	                ///////////// 1660: chiusura chela lato 2 (HMI)
	            1660:
	                "DB_RobotMission".Gripper_Side := 2;
	                "DB_RobotMission".Gripper_code := #Gripper_ID[2];
	                "DB_RobotMission".Command := "CMD_RobotCloseGripper2";
	                #Dispatcher["_master"] := 1661;
	            1661:
	                IF "DB_RobotMissionStatus".StatusCode = "cmd_acquired" OR
	                    "DB_RobotMissionStatus".StatusCode = "cmd_executing" THEN
	                    #Dispatcher["_master"] := 1662;
	                END_IF;
	            1662:
	                IF "DB_RobotMissionStatus".StatusCode = "cmd_executed" THEN
	                    "DB_RobotMission".Command := 0;
	                    #MissionCode := 0;
	                    #Dispatcher["_master"] := 0;
	                END_IF;
	                ///////////// 1700: posizionamento davanti a MC1 (automatico)
	                // Il robot si porta in attesa e la missione chiude: restera' fermo
	                // li' perche' FB204 non assegna nulla finche' la porta non si apre.
	            1700:
	                IF "DB_RobotMissionStatus".StatusCode = "cmd_acquired" OR
	                    "DB_RobotMissionStatus".StatusCode = "cmd_executing" THEN
	                    #Dispatcher["_master"] := 1701;
	                ELSIF "DB_RobotMissionStatus".StatusCode = "cmd_rejected" OR
	                    "DB_RobotMissionStatus".StatusCode = "cmd_aborted" THEN
	                    "DB_RobotMission".Command := 0;
	                    #Error := "MISSION_PositioningMC_AUTO" * 100 + 22;
	                    #MissionCode := 0;
	                    #Dispatcher["_master"] := 0;
	                END_IF;
	            1701:
	                IF "DB_RobotMissionStatus".StatusCode = "cmd_executed" THEN
	                    "DB_RobotMission".Command := 0;
	                    #MissionCode := 0;
	                    #Dispatcher["_master"] := 0;
	                END_IF;
	                ///////////// 1750: ritorno in home (automatico)
	                // Stessa struttura del 1700: attesa acquisizione con gestione del
	                // rifiuto, poi attesa esecuzione. Il robot ci va e resta li'.
	            1750:
	                IF "DB_RobotMissionStatus".StatusCode = "cmd_acquired" OR
	                    "DB_RobotMissionStatus".StatusCode = "cmd_executing" THEN
	                    #Dispatcher["_master"] := 1751;
	                ELSIF "DB_RobotMissionStatus".StatusCode = "cmd_rejected" OR
	                    "DB_RobotMissionStatus".StatusCode = "cmd_aborted" THEN
	                    // il robot non ha accettato: si chiude comunque. Il home e' una
	                    // rifinitura, non deve fermare la cella se fallisce.
	                    "DB_RobotMission".Command := 0;
	                    #MissionCode := 0;
	                    #Dispatcher["_master"] := 0;
	                END_IF;
	            1751:
	                IF "DB_RobotMissionStatus".StatusCode = "cmd_executed" THEN
	                    "DB_RobotMission".Command := 0;
	                    #MissionCode := 0;
	                    #Dispatcher["_master"] := 0;
	                END_IF;
	        END_CASE;
	    END_IF;

	END_REGION

	REGION Gripper_MANAGER
	    REGION Gripper_Robot_to_TRAY
	        CASE #Dispatcher["_Gripper_Robot_to_TRAY"] OF
	            0:  //nothing to do
	                ;
	            10:  //prepare mission data
	                IF "SqlCommands".sqlCommands[0] = '' THEN
	                    IF NOT "DB_BOX_1".Robot_enabled_to_work THEN
	                        #Error := 949;
	                        #Dispatcher["_Gripper_Robot_to_TRAY"] := 0;
	                    ELSE
	                        #queryTemp := CONCAT(IN1 := 'SELECT X,Y,Z,X_ROT,Y_ROT,Z_ROT,APPROACH_TYPE,APPROACH_X,APPROACH_Y,APPROACH_Z from COORDINATES_GRIPPER_SHELF where id=',
	                                             IN2 := "INT_TO_STRING_WITHOUT_SIGN"(#Gripper_ID[1]));
	                        #queryStartExecution := TRUE;

	                        #Dispatcher["_Gripper_Robot_to_TRAY"] := 20;
	                    END_IF;
	                END_IF;

	            20:  // wait for result DB -> prepare mission data
	                // PRESA IN CARICO VERIFICATA: SqlData e' un buffer unico condiviso,
	                // senza il confronto su sqlCommands[0] si legge la risposta di un
	                // altro richiedente — qui sarebbe lo SLOT A SCAFFALE dove posare
	                // la pinza.
	                IF NOT "DB_executeQuery".readyForNextQuery
	                    AND "SqlCommands".sqlCommands[0] = #queryTemp THEN
	                    #Dispatcher["_Gripper_Robot_to_TRAY"] := 25;
	                END_IF;

	            25: //execute query
	                IF "DB_executeQuery".dataReady AND "DB_executeQuery".noData THEN
	                    // slot di casa della pinza non trovato a scaffale: con FB6
	                    // corretto "zero righe" non e' piu' dataError, va preso qui.
	                    #Error := 990;
	                    "DB_executeQuery".readyForNextQuery := TRUE;
	                    #Dispatcher["_Gripper_Robot_to_TRAY"] := 990;
	                ELSIF "DB_executeQuery".dataReady AND NOT "DB_executeQuery".dataError THEN

	                    "DB_RobotMission".Command := "CMD_RobotRemoveGripper";
	                    "DB_RobotMission"."X_Pick-Place" := "SqlData".data.rows[0].col[0];
	                    "DB_RobotMission"."Y_Pick-Place" := "SqlData".data.rows[0].col[1];
	                    "DB_RobotMission"."Z_Pick-Place" := "SqlData".data.rows[0].col[2];
	                    "DB_RobotMission"."XRot_Pick-Place" := "SqlData".data.rows[0].col[3];
	                    "DB_RobotMission"."YRot_Pick-Place" := "SqlData".data.rows[0].col[4];
	                    "DB_RobotMission"."ZRot_Pick-Place" := "SqlData".data.rows[0].col[5];
	                    "DB_RobotMission".X_approach := "SqlData".data.rows[0].col[7];
	                    "DB_RobotMission".Y_approach := "SqlData".data.rows[0].col[8];
	                    "DB_RobotMission".Z_approach := "SqlData".data.rows[0].col[9];
	                    "DB_RobotMission".XRot_approach := 0;
	                    "DB_RobotMission".YRot_approach := 0;
	                    "DB_RobotMission".ZRot_approach := 0;
	                    //"DB_RobotMission".ApproachType := DINT_TO_INT("SqlData".data.rows[0].col[6]);
	                    "DB_RobotMission".ApproachType := "FC_ExtractApproach"(approachVal := "SqlData".data.rows[0].col[6], pick := FALSE);
	                    "DB_RobotMission".Object_Type := "Gripper";
	                    "DB_RobotMission".Unit_code := "Warehouse1";
	                    "DB_RobotMission".Gripper_code := #Gripper_ID[1];
	                    //"DB_RobotMission".Option

	                    "DB_executeQuery".readyForNextQuery := TRUE;

	                    #Dispatcher["_Gripper_Robot_to_TRAY"] := 30;
	                ELSIF "DB_executeQuery".dataError THEN
	                    // Alarm
	                    #Error := 990;
	                    "DB_executeQuery".readyForNextQuery := TRUE;

	                    #Dispatcher["_Gripper_Robot_to_TRAY"] := 990;
	                END_IF;
	            30:  // start robot mission
	                //"DB_RobotMission".Command := "CMD_RobotRemoveGripper";
	                IF "DB_RobotMissionStatus".StatusCode = "cmd_acquired" OR
	                    "DB_RobotMissionStatus".StatusCode = "cmd_executing" THEN
	                    #Dispatcher["_Gripper_Robot_to_TRAY"] := 40;
	                END_IF;
	            40:  // finished -> update DB
	                // DOPPIA CONFERMA (5/9), simmetrica a quella del carico allo
	                // stato 50 di Gripper_TRAY_to_Robot: non basta cmd_executed del
	                // robot, serve anche che il sensore NON veda piu' la pinza.
	                // Senza, i registri direbbero "flangia nuda" con la pinza ancora
	                // attaccata, e ogni scelta successiva partirebbe da un dato falso.
	                // Stallo qui = guardare %I502.0.
	                // NB: lo scarico NON passa dalla catena unica — azzerare i registri
	                // e' un gesto che non ha bisogno di cercare gemelle, e #GripperRequested
	                // deve restare intatto per il carico che i rami 110/210/310/410/510
	                // lanciano subito dopo.
	                IF "DB_RobotMissionStatus".StatusCode = "cmd_executed"
	                    AND NOT "Gripper_mounted"
	                THEN
	                    "DB_RobotMission".Command := 0;  ///\\\
	                    #Gripper_ID[1] := 0;
	                    #Gripper_ID[2] := 0;
	                    #Dispatcher["updateGripperOnRobot"] := 10;

	                    #Dispatcher["_Gripper_Robot_to_TRAY"] := 50;
	                END_IF;
	            50: // attesa fine update DB -> chiusura catena scarico
	                IF #Dispatcher["updateGripperOnRobot"] = 0 THEN
	                    #Dispatcher["_Gripper_Robot_to_TRAY"] := 0;
	                END_IF;

	        END_CASE;
	    END_REGION

	    REGION Gripper_TRAY_to_Robot
	        CASE #Dispatcher["_Gripper_TRAY_to_Robot"] OF
	            0: // nothing to do
	                ;
	            10: //prepare mission data
	                IF "SqlCommands".sqlCommands[0] = '' THEN
	                    IF NOT "DB_BOX_1".Robot_enabled_to_work THEN
	                        #Error := 949;
	                        #Dispatcher["_Gripper_TRAY_to_Robot"] := 0;
	                    ELSE
	                        // SORGENTE UNICA: #GripperRequested (17/9).
	                        // Prima i tre rami leggevano sorgenti diverse — GripperRequested
	                        // per il magazzino, order.GRIPPER per MC1, order.GRIPPER di MC1
	                        // anche nel ramo MC2 (refuso). Nel ciclo automatico i valori
	                        // coincidono perche' i master 100/300/400/500 scrivono
	                        // GripperRequested := order.GRIPPER prima di lanciare, ma
	                        // l'accoppiamento era implicito: la catena cercava a scaffale
	                        // una pinza e la catena unica ne registrava un'altra se le due
	                        // sorgenti divergevano.
	                        // Adesso chi lancia dice QUALE pinza vuole, e questa catena
	                        // la cerca e basta — stessa variabile che _Set_Gripper_OnBoard
	                        // usera' per scrivere i registri.
	                        IF #GripperRequested > 0 THEN
	                            // GEMELLA SOLO CON SUB_POS VALORIZZATO (5/10, concordato 1/9): una pinza
	                            // singola ha SUB_POS = 0, e "SUB_POS in (0)" tirava dentro tutte le altre
	                            // pinze singole a scaffale come se fossero il suo lato 2.
	                            #queryTemp := CONCAT_STRING(IN1 := 'select X,Y,Z,X_rot,Y_rot,Z_ROT, APPROACH_TYPE, APPROACH_X, APPROACH_Y, APPROACH_Z, ID from COORDINATES_GRIPPER_SHELF where id=',
	                                                        IN2 := "INT_TO_STRING_WITHOUT_SIGN"(#GripperRequested),
	                                                        IN3 := ' OR (SUB_POS>0 AND SUB_POS in (select sub_pos from COORDINATES_GRIPPER_SHELF where id=',
	                                                        IN4 := "INT_TO_STRING_WITHOUT_SIGN"(#GripperRequested),
	                                                        IN5 := ')) order by gripper_sub_pos');
	                            #queryStartExecution := TRUE;
	                            #Dispatcher["_Gripper_TRAY_to_Robot"] := 20;
	                        ELSE
	                            // nessuna pinza richiesta: senza questa guardia la query
	                            // usciva con id=0, zero righe e 990 — lo stesso difetto
	                            // che il 17/9 ha tenuto appeso il master ai rami 1xx.
	                            #Error := 937;   // pinza target non valida
	                            #Dispatcher["_Gripper_TRAY_to_Robot"] := 0;
	                        END_IF;
	                    END_IF;
	                END_IF;

	            20:  //execute query
	                // PRESA IN CARICO VERIFICATA: SqlData e' un buffer unico condiviso,
	                // senza il confronto su sqlCommands[0] si legge la risposta di un
	                // altro richiedente — qui sarebbe lo SLOT della pinza da prendere.
	                IF NOT "DB_executeQuery".readyForNextQuery
	                    AND "SqlCommands".sqlCommands[0] = #queryTemp THEN
	                    #Dispatcher["_Gripper_TRAY_to_Robot"] := 30;
	                END_IF;

	            30: // wait anwser
	                IF "DB_executeQuery".dataReady AND "DB_executeQuery".noData THEN
	                    // pinza richiesta non trovata a scaffale. Ramo NUOVO: prima
	                    // non esisteva, e con FB6 corretto la catena proseguirebbe
	                    // con coordinate a zero mandando il robot a sbattere.
	                    #Error := 990;
	                    "DB_executeQuery".readyForNextQuery := true;
	                    #Dispatcher["_Gripper_TRAY_to_Robot"] := 0;
	                ELSIF "DB_executeQuery".dataReady AND NOT "DB_executeQuery".dataError THEN
	                    "DB_RobotMission"."X_Pick-Place" := "SqlData".data.rows[0].col[0];
	                    "DB_RobotMission"."Y_Pick-Place" := "SqlData".data.rows[0].col[1];
	                    "DB_RobotMission"."Z_Pick-Place" := "SqlData".data.rows[0].col[2];
	                    "DB_RobotMission"."XRot_Pick-Place" := "SqlData".data.rows[0].col[3];
	                    "DB_RobotMission"."YRot_Pick-Place" := "SqlData".data.rows[0].col[4];
	                    "DB_RobotMission"."ZRot_Pick-Place" := "SqlData".data.rows[0].col[5];
	                    "DB_RobotMission".X_approach := "SqlData".data.rows[0].col[7];
	                    "DB_RobotMission".Y_approach := "SqlData".data.rows[0].col[8];
	                    "DB_RobotMission".Z_approach := "SqlData".data.rows[0].col[9];
	                    "DB_RobotMission".XRot_approach := 0;
	                    "DB_RobotMission".YRot_approach := 0;
	                    "DB_RobotMission".ZRot_approach := 0;
	                    //"DB_RobotMission".ApproachType := DINT_TO_INT("SqlData".data.rows[0].col[6]);
	                    "DB_RobotMission".ApproachType := "FC_ExtractApproach"(approachVal := "SqlData".data.rows[0].col[6], pick := TRUE);
	                    "DB_RobotMission".Object_Type := "Gripper";
	                    "DB_RobotMission".Unit_code := "Warehouse1";
	                    "DB_RobotMission".Gripper_code := DINT_TO_INT(#GripperRequested);
	                    //"DB_RobotMission".Option

	                    // LATO 2 NON PIU' QUI (17/9): lo scrive la catena
	                    // _Set_Gripper_OnBoard, che e' il punto unico. Questo stato
	                    // leggeva le coordinate di prelievo e per comodita' anche la
	                    // gemella, ma quella doppia responsabilita' e' proprio il
	                    // motivo per cui lo swap — che non passa di qui — dimenticava
	                    // il lato 2.

	                    "DB_executeQuery".readyForNextQuery := true;

	                    #Dispatcher["_Gripper_TRAY_to_Robot"] := 40;
	                ELSIF "DB_executeQuery".dataError THEN
	                    // ramo NUOVO: errore vero del ponte
	                    #Error := 990;
	                    "DB_executeQuery".readyForNextQuery := true;
	                    #Dispatcher["_Gripper_TRAY_to_Robot"] := 0;
	                END_IF;

	            40:  // start Robot mission
	                IF "DB_RobotMissionStatus".StatusCode = "cmd_executed" OR
	                    "DB_RobotMissionStatus".StatusCode = "cmd_waitingNewCmd" THEN
	                    "DB_RobotMission".Command := "CMD_RobotPickGripper";

	                    #Dispatcher["_Gripper_TRAY_to_Robot"] := 45;
	                END_IF;
	            45:
	                //"DB_RobotMission".Command := "CMD_RobotPickGripper";
	                IF "DB_RobotMissionStatus".StatusCode = "cmd_acquired" OR
	                    "DB_RobotMissionStatus".StatusCode = "cmd_executing" THEN

	                    #Dispatcher["_Gripper_TRAY_to_Robot"] := 50;
	                END_IF;

	            50: // latch a doppia conferma: esito missione + sensore fisico — stallo qui = guardare %I502.0
	                IF "DB_RobotMissionStatus".StatusCode = "cmd_executed" AND "Gripper_mounted" THEN

	                    // AZZERAMENTO COMANDO (5/9): senza, il robot resta a
	                    // cmd_executed in attesa che il PLC risponda, e get_TCP_Data
	                    // allo stato 40 aspetta che il robot torni a waitingNewCmd:
	                    // stallo circolare col master fermo al 960.
	                    "DB_RobotMission".Command := 0;  ///\\\

	                    // registri + database alla catena unica (17/9)
	                    #Dispatcher["_Set_Gripper_OnBoard"] := 10;
	                    #Dispatcher["_Gripper_TRAY_to_Robot"] := 60;
	                END_IF;
	            60: // attesa fine registrazione -> chiusura catena carico
	                IF #Dispatcher["_Set_Gripper_OnBoard"] = 0 THEN
	                    #Dispatcher["_Gripper_TRAY_to_Robot"] := 0;
	                END_IF;
	        END_CASE;

	    END_REGION

	    REGION Gripper_Hook_Search
	        CASE #Dispatcher["_Gripper_Hook_Search"] OF
	            0: // nothing to do
	                ;
	            10: //prepare mission data
	                IF "SqlCommands".sqlCommands[0] = '' THEN
	                    //#queryTemp := 'select id,pos_mag-1000 from gripper where pos_mag>1000 and pos_plant>=0';
	                    #queryTemp := 'select id,sub_pos-1000 from gripper where sub_pos>1000 AND pos_plant>=0';
	                    #queryStartExecution := TRUE;
	                    #Dispatcher["_Gripper_Hook_Search"] := 20;
	                END_IF;

	            20:  //execute query
	                // PRESA IN CARICO VERIFICATA: SqlData e' un buffer unico condiviso,
	                // senza il confronto su sqlCommands[0] si legge la risposta di un
	                // altro richiedente — qui finirebbe in GripperRequested un ID pinza
	                // preso da una colonna qualsiasi di un'altra query.
	                IF NOT "DB_executeQuery".readyForNextQuery
	                    AND "SqlCommands".sqlCommands[0] = #queryTemp THEN
	                    #Dispatcher["_Gripper_Hook_Search"] := 30;
	                END_IF;

	            30: // wait anwser
	                IF "DB_executeQuery".dataReady THEN
	                    IF "DB_executeQuery".noData OR "DB_executeQuery".dataError THEN
	                        #Error := 22;
	                    ELSE
	                        #GripperRequested := DINT_TO_INT("SqlData".data.rows[0].col[1]);
	                    END_IF;

	                    "DB_executeQuery".readyForNextQuery := true;
	                    #Dispatcher["_Gripper_Hook_Search"] := 0;
	                END_IF;
	        END_CASE;

	    END_REGION

	    REGION Gripper4Pallet_Search
	        CASE #Dispatcher["_Gripper4Pallet_Search"] OF
	            0: // nothing to do
	                ;
	            10: //prepare mission data
	                IF "SqlCommands".sqlCommands[0] = '' THEN
	                    #queryTemp := CONCAT_STRING(IN1 := 'select GRIPPERREQ from pallets_grippers where palletID=',
	                                                IN2 := "INT_TO_STRING_WITHOUT_SIGN"(#PalletRequested));
	                    #queryStartExecution := TRUE;
	                    #Dispatcher["_Gripper4Pallet_Search"] := 20;
	                END_IF;

	            20:  //execute query
	                // PRESA IN CARICO VERIFICATA: SqlData e' un buffer unico condiviso,
	                // senza il confronto su sqlCommands[0] si legge la risposta di un
	                // altro richiedente — qui finirebbe in GripperRequested un ID pinza
	                // preso da una colonna qualsiasi di un'altra query.
	                IF NOT "DB_executeQuery".readyForNextQuery
	                    AND "SqlCommands".sqlCommands[0] = #queryTemp THEN
	                    #Dispatcher["_Gripper4Pallet_Search"] := 30;
	                END_IF;

	            30: // wait anwser
	                IF "DB_executeQuery".dataReady THEN
	                    IF "DB_executeQuery".noData OR "DB_executeQuery".dataError THEN
	                        #Error := "_Gripper4Pallet_Search" * 100 + 22;
	                    ELSE
	                        #GripperRequested := DINT_TO_INT("SqlData".data.rows[0].col[0]);
	                    END_IF;

	                    "DB_executeQuery".readyForNextQuery := true;
	                    #Dispatcher["_Gripper4Pallet_Search"] := 0;
	                END_IF;
	        END_CASE;
	    END_REGION

	    REGION Set_Gripper_OnBoard
	        // PUNTO UNICO DI SCRITTURA DEI REGISTRI PINZA (17/9).
	        // Prima Gripper_ID[1] e [2] venivano scritti da piu' percorsi diversi e
	        // ognuno doveva ricordarsi di cercare la gemella: lo swap non lo faceva,
	        // e siccome il 35 di FB204 cambia pinza SEMPRE via swap, in automatico il
	        // lato 2 restava a zero e la pinza doppia veniva usata come singola.
	        // Da qui in poi chi monta una pinza scrive #GripperRequested e lancia
	        // questa catena: la gemella la cerca lei, i registri li scrive lei, il
	        // database lo allinea lei.
	        //
	        // INGRESSO:  #GripperRequested = ID pinza a bordo, 0 = flangia nuda
	        // USCITA:    Gripper_ID[1], Gripper_ID[2], POS_PLANT a database
	        //
	        // La query e' sulla TABELLA GRIPPER, non sulla vista dello scaffale:
	        // la vista puo' non contenere una pinza gia' registrata a bordo.
	        CASE #Dispatcher["_Set_Gripper_OnBoard"] OF
	            0: // nothing to do
	                ;

	            10: // flangia nuda oppure ricerca gemella
	                IF #GripperRequested <= 0 THEN
	                    #Gripper_ID[1] := 0;
	                    #Gripper_ID[2] := 0;
	                    #Dispatcher["updateGripperOnRobot"] := 10;
	                    #Dispatcher["_Set_Gripper_OnBoard"] := 50;
	                ELSIF "SqlCommands".sqlCommands[0] = '' THEN
	                    #queryTemp := CONCAT(IN1 := 'select ID from GRIPPER where ID=',
	                                         IN2 := "INT_TO_STRING_WITHOUT_SIGN"(#GripperRequested),
	                                         IN3 := ' or (SUB_POS>0 and SUB_POS in (select SUB_POS from GRIPPER where ID=',
	                                         IN4 := "INT_TO_STRING_WITHOUT_SIGN"(#GripperRequested),
	                                         IN5 := '))');
	                    #queryStartExecution := TRUE;
	                    #Dispatcher["_Set_Gripper_OnBoard"] := 20;
	                END_IF;

	            20: // presa in carico VERIFICATA
	                IF NOT "DB_executeQuery".readyForNextQuery
	                    AND "SqlCommands".sqlCommands[0] = #queryTemp THEN
	                    #Dispatcher["_Set_Gripper_OnBoard"] := 30;
	                END_IF;

	            30: // esito: due righe = pinza doppia, la gemella e' il lato 2.
	                // La query include se stessa, quindi una riga sola significa
	                // pinza singola. Su errore o zero righe NON si alza allarme: la
	                // pinza e' fisicamente a bordo e il ciclo deve poter proseguire
	                // come singola — che e' il comportamento storico.
	                IF "DB_executeQuery".dataReady THEN
	                    #Gripper_ID[1] := #GripperRequested;
	                    #Gripper_ID[2] := 0;

	                    IF NOT "DB_executeQuery".noData
	                        AND NOT "DB_executeQuery".dataError
	                        AND "SqlData".data.rowCount > 1
	                    THEN
	                        IF DINT_TO_INT("SqlData".data.rows[0].col[0]) <> #GripperRequested THEN
	                            #Gripper_ID[2] := DINT_TO_INT("SqlData".data.rows[0].col[0]);
	                        ELSE
	                            #Gripper_ID[2] := DINT_TO_INT("SqlData".data.rows[1].col[0]);
	                        END_IF;
	                    END_IF;

	                    "DB_executeQuery".readyForNextQuery := TRUE;
	                    #queryTemp := '';
	                    #queryStartExecution := FALSE;

	                    #Dispatcher["updateGripperOnRobot"] := 10;
	                    #Dispatcher["_Set_Gripper_OnBoard"] := 50;
	                END_IF;

	            50: // allineamento database chiuso
	                IF #Dispatcher["updateGripperOnRobot"] = 0 THEN
	                    #Dispatcher["_Set_Gripper_OnBoard"] := 0;
	                END_IF;
	        END_CASE;
	    END_REGION

	END_REGION

	REGION PALLETS_MANAGER
	    REGION Pallet_Tray_to_Robot
	        CASE #Dispatcher["_Pallet_TRAY_to_Robot"] OF
	            0: //nothing to do
	                ;
	            10: //prepare mission data
	                IF "SqlCommands".sqlCommands[0] = '' THEN
	                    IF #GripperOccuped[1] THEN
	                        //gripper occupata
	                        #Error := 21;
	                        #Dispatcher["_Pallet_TRAY_to_Robot"] := 0;
	                    ELSIF #MCRequested = 1 AND "DB_MC1".order.ID <= 0 THEN
	                        #Error := "_Pallet_TRAY_to_Robot" * 1000 + 1;  //Error 1001
	                        #Dispatcher["_Pallet_TRAY_to_Robot"] := "_Pallet_TRAY_to_Robot" * 1000 + 1;
	                    ELSIF #MCRequested = 2 AND "DB_MC2".order.ID <= 0 THEN
	                        #Error := "_Pallet_TRAY_to_Robot" * 1000 + 2;  //Erroe 1002
	                        #Dispatcher["_Pallet_TRAY_to_Robot"] := "_Pallet_TRAY_to_Robot" * 1000 + 2;
	                    ELSIF #RemoteMode AND #MCRequested = 1 THEN
	                        #queryTemp := CONCAT(IN1 := 'select * from COORDINATES_FOR_PALLET_WAREHOUSE  where status=4 and palletID = ',  //Order_ID
	                                             IN2 := "INT_TO_STRING_WITHOUT_SIGN"(DINT_TO_INT("DB_MC1".order.PALLET)));
	                        #queryStartExecution := TRUE;
	                        #Dispatcher["_Pallet_TRAY_to_Robot"] := 20;
	                    ELSIF #RemoteMode AND #MCRequested = 2 THEN
	                        #queryTemp := CONCAT(IN1 := 'select * from COORDINATES_FOR_PALLET_WAREHOUSE  where status=4 and PalletID = ',  //Order_ID
	                                             IN2 := "INT_TO_STRING_WITHOUT_SIGN"(DINT_TO_INT("DB_MC2".order.PALLET)));
	                        #queryStartExecution := TRUE;
	                        #Dispatcher["_Pallet_TRAY_to_Robot"] := 20;
	                    ELSIF NOT #RemoteMode AND #MCRequested = 0 THEN  //COMMAND FROM HMI
	                        #queryTemp := CONCAT(IN1 := 'select * from COORDINATES_FOR_PALLET_WAREHOUSE where POS= ',
	                                             IN2 := "INT_TO_STRING_WITHOUT_SIGN"(DINT_TO_INT(#PalletPosition)));
	                        #queryStartExecution := TRUE;
	                        #Dispatcher["_Pallet_TRAY_to_Robot"] := 20;
	                    END_IF;
	                END_IF;

	            20:  //execute query
	                // PRESA IN CARICO VERIFICATA: SqlData e' un buffer unico condiviso,
	                // senza il confronto su sqlCommands[0] si legge la risposta di un
	                // altro richiedente — qui sarebbero le COORDINATE del pallet a
	                // magazzino, comprese le rotazioni di approccio.
	                IF NOT "DB_executeQuery".readyForNextQuery
	                    AND "SqlCommands".sqlCommands[0] = #queryTemp THEN
	                    #Dispatcher["_Pallet_TRAY_to_Robot"] := 30;
	                END_IF;

	            30:  // wait for result DB -> prepare mission data
	                IF "DB_executeQuery".dataReady AND "DB_executeQuery".noData THEN
	                    // nessun pallet pronto: con FB6 corretto "zero righe" non e'
	                    // piu' dataError, va intercettato qui.
	                    "DB_executeQuery".readyForNextQuery := TRUE;

	                    #Error := "_Pallet_TRAY_to_Robot" * 1000 + 10;  //Error 1010
	                    #Dispatcher["_Pallet_TRAY_to_Robot"] := "_Pallet_TRAY_to_Robot" * 1000 + 10;
	                ELSIF "DB_executeQuery".dataReady AND NOT "DB_executeQuery".dataError THEN
	                    "DB_RobotMission"."X_Pick-Place" := ("SqlData".data.rows[0].col[0]);
	                    "DB_RobotMission"."Y_Pick-Place" := ("SqlData".data.rows[0].col[1]);
	                    "DB_RobotMission"."Z_Pick-Place" := ("SqlData".data.rows[0].col[2]);
	                    "DB_RobotMission"."XRot_Pick-Place" := ("SqlData".data.rows[0].col[3]);
	                    "DB_RobotMission"."YRot_Pick-Place" := ("SqlData".data.rows[0].col[4]);
	                    "DB_RobotMission"."ZRot_Pick-Place" := ("SqlData".data.rows[0].col[5]);
	                    "DB_RobotMission".X_approach := ("SqlData".data.rows[0].col[6]);
	                    "DB_RobotMission".Y_approach := ("SqlData".data.rows[0].col[7]);
	                    "DB_RobotMission".Z_approach := ("SqlData".data.rows[0].col[8]);
	                    "DB_RobotMission".XRot_approach := ("SqlData".data.rows[0].col[9]);
	                    "DB_RobotMission".YRot_approach := ("SqlData".data.rows[0].col[10]);
	                    "DB_RobotMission".ZRot_approach := ("SqlData".data.rows[0].col[11]);
	                    //"DB_RobotMission".ApproachType := DINT_TO_INT("SqlData".data.rows[0].col[12]);
	                    "DB_RobotMission".ApproachType := "FC_ExtractApproach"(approachVal := "SqlData".data.rows[0].col[12], pick := TRUE);
	                    "DB_RobotMission".Object_Type := "Pallet";
	                    "DB_RobotMission".Unit_code := "WarehousePallet";
	                    "DB_RobotMission".Gripper_code := #GripperRequested;
	                    "DB_RobotMission".Gripper_Side := 1;
	                    //"DB_RobotMission".Option

	                    "DB_executeQuery".readyForNextQuery := TRUE;

	                    #Dispatcher["_Pallet_TRAY_to_Robot"] := 40;
	                ELSIF "DB_executeQuery".dataError THEN
	                    "DB_executeQuery".readyForNextQuery := TRUE;

	                    #Error := "_Pallet_TRAY_to_Robot" * 1000 + 10;  //Error 1010
	                    #Dispatcher["_Pallet_TRAY_to_Robot"] := "_Pallet_TRAY_to_Robot" * 1000 + 10;
	                END_IF;
	            40:
	                "DB_RobotMission".Command := "CMD_RobotPickObject";
	                IF "DB_RobotMissionStatus".StatusCode = "cmd_acquired" OR
	                    "DB_RobotMissionStatus".StatusCode = "cmd_executing" THEN

	                    #Dispatcher["_Pallet_TRAY_to_Robot"] := 50;
	                END_IF;
	            50:
	                IF "DB_RobotMissionStatus".StatusCode = "cmd_executed" THEN
	                    "DB_RobotMission".Command := 0;  ///\\\
	                    #GripperOccuped[1] := TRUE;
	                    #Dispatcher["updatePartOnRobot"] := 10 + DINT_TO_INT("RAW");  //il pallet lo considero grezzo cosi va in macchina

	                    #Dispatcher["_Pallet_TRAY_to_Robot"] := 60;
	                END_IF;
	            60:  // updateDB
	                IF #Dispatcher["updatePartOnRobot"] = 0 THEN
	                    #Dispatcher["updatePalletOnTRAY"] := 10 + DINT_TO_INT("EMPTY");

	                    #Dispatcher["_Pallet_TRAY_to_Robot"] := 70;
	                END_IF;
	            70:
	                IF #Dispatcher["updatePalletOnTRAY"] = 0 THEN
	                    #Dispatcher["_Pallet_TRAY_to_Robot"] := 0;
	                END_IF;

	                // ==== ERRORS 1xxx ====
	            1001:
	                ; //WorkOrder not defined for MC1
	            1002:
	                ; //WorkOrder not defined for MC2
	            1010:
	                ; //No pallets ready for work
	                // ==== ERRORS 1xxx ====

	        END_CASE;
	    END_REGION

	    REGION Pallet_Robot_to_Tray
	        CASE #Dispatcher["_Pallet_Robot_to_TRAY"] OF
	            0: //nothing to do
	                ;
	            10: //prepare mission data
	                IF "SqlCommands".sqlCommands[0] = '' THEN
	                    IF NOT #GripperOccuped[1] AND "Gripper1_Closed" THEN   //non usare direttamente Ingresso
	                        //gripper empty
	                        #Error := 2021;
	                        #Dispatcher["_Pallet_Robot_to_TRAY"] := 2021;
	                    ELSIF #MCRequested = 1 AND "DB_MC1".order.ID <= 0 THEN
	                        #Error := 2001;
	                        #Dispatcher["_Pallet_Robot_to_TRAY"] := 2001;
	                    ELSIF #MCRequested = 2 AND "DB_MC2".order.ID <= 0 THEN
	                        #Error := 2002;
	                        #Dispatcher["_Pallet_Robot_to_TRAY"] := 2002;
	                    ELSIF #MCRequested = 1 THEN
	                        #queryTemp := CONCAT(IN1 := 'select * from COORDINATES_FOR_PALLET_WAREHOUSE where PalletID = ',  //Order_ID
	                                             IN2 := "INT_TO_STRING_WITHOUT_SIGN"(DINT_TO_INT("DB_MC1".order.PALLET)),
	                                             IN3 := ' AND Status=2');
	                        #queryStartExecution := TRUE;
	                        #Dispatcher["_Pallet_Robot_to_TRAY"] := 20;
	                    ELSIF #MCRequested = 2 THEN
	                        #queryTemp := CONCAT(IN1 := 'select * from COORDINATES_FOR_PALLET_WAREHOUSE where PalletID = ',
	                                             IN2 := "INT_TO_STRING_WITHOUT_SIGN"(DINT_TO_INT("DB_MC2".order.PALLET)),
	                                             IN3 := ' AND Status=2');
	                        #queryStartExecution := TRUE;
	                        #Dispatcher["_Pallet_Robot_to_TRAY"] := 20;
	                    ELSIF #MCRequested = 0 THEN     //HMI COMMAND
	                        // VISTA NUOVA (16/9): COORDINATES_FOR_PALLET_WAREHOUSE e' un
	                        // join implicito fra POSITION e PALLET su sub_pos = MAG_POS,
	                        // quindi restituisce SOLO i posti gia' occupati — le venti
	                        // posizioni libere non ci sono per costruzione, e il deposito
	                        // in un posto vuoto dava 2005 (visto 16/9).
	                        // Il join non era un errore: la Y dipende dalle misure del
	                        // pallet (Y/2, Y_CORR, Y_HandlePoint), quindi una posizione
	                        // senza pallet non ha coordinate calcolabili. Serviva la
	                        // combinazione POSTO x PALLET, che e' COORDINATES_FOR_PALLET_PLACE:
	                        // stesso calcolo, CROSS JOIN, filtrata sui due parametri.
	                        // Verificato che sul posto 10 col pallet 9 le due viste danno
	                        // le stesse identiche coordinate.
	                        #queryTemp := CONCAT(IN1 := 'select X,Y,Z,X_ROT,Y_ROT,Z_ROT,APPROACH_X,APPROACH_Y,APPROACH_Z,APPROACH_X_ROT,APPROACH_Y_ROT,APPROACH_Z_ROT,APPROACH_TYPE from COORDINATES_FOR_PALLET_PLACE where POS=',
	                                             IN2 := "INT_TO_STRING_WITHOUT_SIGN"(DINT_TO_INT(#PalletPosition)),
	                                             IN3 := ' and PalletID=',
	                                             IN4 := "INT_TO_STRING_WITHOUT_SIGN"(#PalletRequested));
	                        #queryStartExecution := TRUE;
	                        #Dispatcher["_Pallet_Robot_to_TRAY"] := 20;
	                    END_IF;
	                END_IF;

	            20:  //execute query
	                // PRESA IN CARICO VERIFICATA: SqlData e' un buffer unico condiviso,
	                // senza il confronto su sqlCommands[0] si legge la risposta di un
	                // altro richiedente — qui sarebbero le COORDINATE di deposito del
	                // pallet a magazzino.
	                IF NOT "DB_executeQuery".readyForNextQuery
	                    AND "SqlCommands".sqlCommands[0] = #queryTemp THEN
	                    #Dispatcher["_Pallet_Robot_to_TRAY"] := 30;
	                END_IF;

	            30:  // wait for result DB -> prepare mission data
	                IF "DB_executeQuery".dataReady AND "DB_executeQuery".noData THEN
	                    // posizione di deposito pallet non trovata: con FB6 corretto
	                    // "zero righe" non e' piu' dataError, va intercettato qui.
	                    "DB_executeQuery".readyForNextQuery := TRUE;

	                    #Error := 2005;
	                    #Dispatcher["_Pallet_Robot_to_TRAY"] := 2005;
	                ELSIF "DB_executeQuery".dataReady AND NOT "DB_executeQuery".dataError THEN
	                    "DB_RobotMission"."X_Pick-Place" := ("SqlData".data.rows[0].col[0]);
	                    "DB_RobotMission"."Y_Pick-Place" := ("SqlData".data.rows[0].col[1]);
	                    "DB_RobotMission"."Z_Pick-Place" := ("SqlData".data.rows[0].col[2]);
	                    "DB_RobotMission"."XRot_Pick-Place" := ("SqlData".data.rows[0].col[3]);
	                    "DB_RobotMission"."YRot_Pick-Place" := ("SqlData".data.rows[0].col[4]);
	                    "DB_RobotMission"."ZRot_Pick-Place" := ("SqlData".data.rows[0].col[5]);
	                    "DB_RobotMission".X_approach := ("SqlData".data.rows[0].col[6]);
	                    "DB_RobotMission".Y_approach := ("SqlData".data.rows[0].col[7]);
	                    "DB_RobotMission".Z_approach := ("SqlData".data.rows[0].col[8]);
	                    "DB_RobotMission".XRot_approach := ("SqlData".data.rows[0].col[9]);
	                    "DB_RobotMission".YRot_approach := ("SqlData".data.rows[0].col[10]);
	                    "DB_RobotMission".ZRot_approach := ("SqlData".data.rows[0].col[11]);
	                    "DB_RobotMission".ApproachType := "FC_ExtractApproach"(approachVal := "SqlData".data.rows[0].col[12], pick := FALSE);
	                    "DB_RobotMission".Object_Type := "Pallet";
	                    "DB_RobotMission".Unit_code := "WarehousePallet";
	                    "DB_RobotMission".Gripper_code := #GripperRequested;
	                    //"DB_RobotMission".Option

	                    "DB_executeQuery".readyForNextQuery := TRUE;

	                    #Dispatcher["_Pallet_Robot_to_TRAY"] := 40;
	                ELSIF "DB_executeQuery".dataError THEN
	                    "DB_executeQuery".readyForNextQuery := TRUE;

	                    #Error := 2005;
	                    #Dispatcher["_Pallet_Robot_to_TRAY"] := 2005;
	                END_IF;
	            40:
	                "DB_RobotMission".Command := "CMD_RobotPlaceObject";
	                IF "DB_RobotMissionStatus".StatusCode = "cmd_acquired" OR
	                    "DB_RobotMissionStatus".StatusCode = "cmd_executing" THEN

	                    #Dispatcher["_Pallet_Robot_to_TRAY"] := 50;
	                END_IF;
	            50:
	                IF "DB_RobotMissionStatus".StatusCode = "cmd_executed" THEN
	                    "DB_RobotMission".Command := 0;  ///\\\
	                    #GripperOccuped[1] := FALSE;
	                    #Dispatcher["updatePartOnRobot"] := 10 + DINT_TO_INT("EMPTY");

	                    #Dispatcher["_Pallet_Robot_to_TRAY"] := 60;
	                END_IF;
	            60:  // updateDB
	                IF #Dispatcher["updatePartOnRobot"] = 0 THEN
	                    #Dispatcher["updatePalletOnTRAY"] := 10 + DINT_TO_INT("RAW");

	                    #Dispatcher["_Pallet_Robot_to_TRAY"] := 70;
	                END_IF;
	            70:
	                IF #Dispatcher["updatePalletOnTRAY"] = 0 THEN
	                    #Dispatcher["_Pallet_Robot_to_TRAY"] := 0;
	                END_IF;

	        END_CASE;
	    END_REGION

	    REGION Pallet_Robot_to_MC
	        CASE #Dispatcher["_Pallet_Robot_to_MC"] OF
	            0: //nothing to do
	                ;

	            10: //prepare mission data
	                IF "SqlCommands".sqlCommands[0] = '' THEN
	                    IF NOT #GripperOccuped[1] AND NOT #GripperOccuped[2] THEN
	                        //gripper vuota
	                        #Error := 22;
	                        #Dispatcher["_Pallet_Robot_to_MC"] := 3022;
	                    ELSE
	                        IF NOT #RemoteMode THEN
	                            #pieceReq := #PalletRequested;   // comando manuale: pallet dal pannello
	                            IF #pieceReq = 0 THEN
	                                #Error := 936;               // nessun pallet indicato nel comando
	                            END_IF;
	                        ELSE
	                            IF #MCRequested = 1 THEN
	                                #pieceReq := DINT_TO_INT("DB_MC1".order.PALLET);
	                            ELSIF #MCRequested = 2 THEN
	                                #pieceReq := DINT_TO_INT("DB_MC2".order.PALLET);
	                            ELSE
	                                #Error := 936;
	                            END_IF;
	                        END_IF;

	                        IF #Error = 0 THEN
	                            #queryTemp := CONCAT(IN1 := 'select X,Y,Z,X_ROT,Y_ROT,Z_ROT,APPROACH_X,APPROACH_Y,APPROACH_Z,APPROACH_X_ROT, APPROACH_Y_ROT, APPROACH_Z_ROT, APPROACH_TYPE from COORDINATES_MC_FOR_PALLET where parent like $'MC_',
	                                                 IN2 := "INT_TO_STRING_WITHOUT_SIGN"(#MCRequested),
	                                                 IN3 := '_pallet%$' AND SUB_POS=1 AND PalletId=',
	                                                 IN4 := "INT_TO_STRING_WITHOUT_SIGN"(#pieceReq));
	                            #queryStartExecution := true;
	                            #Dispatcher["_Pallet_Robot_to_MC"] := 20;
	                        END_IF;
	                    END_IF;
	                END_IF;

	            20:  //execute query
	                // PRESA IN CARICO VERIFICATA: SqlData e' un buffer unico condiviso,
	                // senza il confronto su sqlCommands[0] si legge la risposta di un
	                // altro richiedente — qui sarebbero le COORDINATE di deposito del
	                // pallet IN MACCHINA.
	                IF NOT "DB_executeQuery".readyForNextQuery
	                    AND "SqlCommands".sqlCommands[0] = #queryTemp THEN
	                    #Dispatcher["_Pallet_Robot_to_MC"] := 30;
	                END_IF;

	            30:  // wait for result DB -> prepare mission data
	                IF "DB_executeQuery".dataReady AND "DB_executeQuery".noData THEN
	                    // posizione pallet in macchina non trovata: con FB6 corretto
	                    // "zero righe" non e' piu' dataError, va intercettato qui.
	                    #Error := 3005;
	                    "DB_executeQuery".readyForNextQuery := TRUE;

	                    #Dispatcher["_Pallet_Robot_to_MC"] := 3005;
	                ELSIF "DB_executeQuery".dataReady AND NOT "DB_executeQuery".dataError THEN

	                    "DB_RobotMission"."X_Pick-Place" := ("SqlData".data.rows[0].col[0]);
	                    "DB_RobotMission"."Y_Pick-Place" := ("SqlData".data.rows[0].col[1]);
	                    "DB_RobotMission"."Z_Pick-Place" := ("SqlData".data.rows[0].col[2]);
	                    "DB_RobotMission"."XRot_Pick-Place" := ("SqlData".data.rows[0].col[3]);
	                    "DB_RobotMission"."YRot_Pick-Place" := ("SqlData".data.rows[0].col[4]);
	                    "DB_RobotMission"."ZRot_Pick-Place" := ("SqlData".data.rows[0].col[5]);
	                    "DB_RobotMission".X_approach := ("SqlData".data.rows[0].col[6]);
	                    "DB_RobotMission".Y_approach := ("SqlData".data.rows[0].col[7]);
	                    "DB_RobotMission".Z_approach := ("SqlData".data.rows[0].col[8]);
	                    "DB_RobotMission".XRot_approach := ("SqlData".data.rows[0].col[9]);
	                    "DB_RobotMission".YRot_approach := ("SqlData".data.rows[0].col[10]);
	                    "DB_RobotMission".ZRot_approach := ("SqlData".data.rows[0].col[11]);
	                    //"DB_RobotMission".ApproachType := DINT_TO_INT("SqlData".data.rows[0].col[12]);
	                    "DB_RobotMission".ApproachType := "FC_ExtractApproach"(approachVal := "SqlData".data.rows[0].col[12], pick := FALSE);
	                    "DB_RobotMission".Object_Type := "Pallet";
	                    "DB_RobotMission".Unit_code := 10 + #MCRequested; //MC1-4 -> 11-14
	                    "DB_RobotMission".Gripper_code := #GripperRequested;
	                    "DB_RobotMission".Gripper_Side := 1;
	                    //"DB_RobotMission".Option
	                    //
	                    "DB_executeQuery".readyForNextQuery := TRUE;

	                    #Dispatcher["_Pallet_Robot_to_MC"] := 40;
	                ELSIF "DB_executeQuery".dataError THEN
	                    //Errore
	                    #Error := 3005;
	                    "DB_executeQuery".readyForNextQuery := TRUE;

	                    #Dispatcher["_Pallet_Robot_to_MC"] := 3005;
	                END_IF;
	            40:
	                "DB_RobotMission".Command := "CMD_RobotPlaceObject";
	                IF "DB_RobotMissionStatus".StatusCode = "cmd_acquired" OR
	                    "DB_RobotMissionStatus".StatusCode = "cmd_executing" THEN
	                    #Dispatcher["_Pallet_Robot_to_MC"] := 50;
	                END_IF;
	            50:
	                IF "DB_RobotMissionStatus".StatusCode = "cmd_executed" THEN
	                    IF "DB_RobotMission".Gripper_Side = 2 THEN
	                        #GripperOccuped[2] := FALSE;
	                    ELSE
	                        #GripperOccuped[1] := FALSE;
	                    END_IF;
	                    "DB_RobotMission".Command := 0;  ///\\\
	                    #Dispatcher["updatePartOnRobot"] := 10 + DINT_TO_INT("EMPTY");

	                    #Dispatcher["_Pallet_Robot_to_MC"] := 60;
	                END_IF;

	            60:
	                IF #Dispatcher["updatePartOnRobot"] = 0 THEN
	                    #Dispatcher["updatePartOnMC"] := 20 + DINT_TO_INT("RAW");

	                    // IL REGISTRO DELLA MACCHINA VA SCRITTO (17/9): simmetrico
	                    // all'azzeramento nel 60 di Pallet_MC_to_Robot. Il pallet e'
	                    // appena entrato; in automatico il 30 substate 2 di FB204 lo
	                    // scrive gia', ma sui comandi MANUALI dal pannello nessuno lo
	                    // faceva e il registro restava a zero.
	                    IF #MCRequested = 1 THEN
	                        "DB_MC1".pallet := #pieceReq;
	                    ELSIF #MCRequested = 2 THEN
	                        "DB_MC2".pallet := #pieceReq;
	                    END_IF;

	                    #Dispatcher["_Pallet_Robot_to_MC"] := 70;
	                END_IF;

	            70:
	                IF #Dispatcher["updatePartOnMC"] = 0 THEN

	                    #Dispatcher["_Pallet_Robot_to_MC"] := 0;
	                END_IF;
	        END_CASE;
	    END_REGION

	    REGION Pallet_MC_to_Robot
	        CASE #Dispatcher["_Pallet_MC_to_Robot"] OF
	            0: //nothing to do
	                ;

	            10: //prepare mission data
	                IF "SqlCommands".sqlCommands[0] = '' THEN
	                    IF #GripperOccuped[1] THEN
	                        #Error := 4022;
	                        #Dispatcher["_Pallet_MC_to_Robot"] := 4022;
	                    ELSIF NOT #RemoteMode THEN   // HMI: pallet esplicito
	                        IF #PalletRequested = 0 THEN
	                            #Error := 936;   // nessun pallet indicato nel comando
	                        ELSE
	                            #queryTemp := CONCAT(IN1 := 'select X,Y,Z,X_ROT,Y_ROT,Z_ROT,APPROACH_X,APPROACH_Y,APPROACH_Z,APPROACH_X_ROT, APPROACH_Y_ROT, APPROACH_Z_ROT, APPROACH_TYPE from COORDINATES_MC_FOR_PALLET where parent like $'MC_',
	                                                 IN2 := "INT_TO_STRING_WITHOUT_SIGN"(#MCRequested),
	                                                 IN3 := '_pallet%$' AND SUB_POS=1 AND PalletID=',
	                                                 IN4 := "INT_TO_STRING_WITHOUT_SIGN"(#PalletRequested));
	                            #queryStartExecution := TRUE;
	                            #Dispatcher["_Pallet_MC_to_Robot"] := 20;
	                        END_IF;
	                    ELSE
	                        #queryTemp := CONCAT(IN1 := 'select X,Y,Z,X_ROT,Y_ROT,Z_ROT,APPROACH_X,APPROACH_Y,APPROACH_Z,APPROACH_X_ROT, APPROACH_Y_ROT, APPROACH_Z_ROT, APPROACH_TYPE from COORDINATES_MC_FOR_PALLET where parent like $'MC_',
	                                             IN2 := "INT_TO_STRING_WITHOUT_SIGN"(#MCRequested),
	                                             IN3 := '_pallet%$' AND SUB_POS=1 AND PalletID=');
	                        IF #MCRequested = 1 THEN
	                            #queryTemp := CONCAT(IN1 := #queryTemp,
	                                                 IN2 := "INT_TO_STRING_WITHOUT_SIGN"(DINT_TO_INT("DB_MC1".order.PALLET)));
	                        ELSE
	                            #Error := 936;
	                        END_IF;

	                        IF #Error = 0 THEN
	                            #queryStartExecution := true;
	                            #Dispatcher["_Pallet_MC_to_Robot"] := 20;
	                        END_IF;
	                    END_IF;
	                END_IF;

	            20:  //execute query
	                // PRESA IN CARICO VERIFICATA: SqlData e' un buffer unico condiviso,
	                // senza il confronto su sqlCommands[0] si legge la risposta di un
	                // altro richiedente — qui sarebbero le COORDINATE di prelievo del
	                // pallet DALLA MACCHINA.
	                IF NOT "DB_executeQuery".readyForNextQuery
	                    AND "SqlCommands".sqlCommands[0] = #queryTemp THEN
	                    #Dispatcher["_Pallet_MC_to_Robot"] := 30;
	                END_IF;

	            30:  // wait for result DB -> prepare mission data
	                IF "DB_executeQuery".dataReady AND "DB_executeQuery".noData THEN
	                    // posizione pallet in macchina non trovata: con FB6 corretto
	                    // "zero righe" non e' piu' dataError, va intercettato qui.
	                    "DB_executeQuery".readyForNextQuery := TRUE;
	                    #Error := 4099;
	                    #Dispatcher["_Pallet_MC_to_Robot"] := 4099;
	                ELSIF "DB_executeQuery".dataReady AND NOT "DB_executeQuery".dataError THEN

	                    "DB_RobotMission"."X_Pick-Place" := ("SqlData".data.rows[0].col[0]);
	                    "DB_RobotMission"."Y_Pick-Place" := ("SqlData".data.rows[0].col[1]);
	                    "DB_RobotMission"."Z_Pick-Place" := ("SqlData".data.rows[0].col[2]);
	                    "DB_RobotMission"."XRot_Pick-Place" := ("SqlData".data.rows[0].col[3]);
	                    "DB_RobotMission"."YRot_Pick-Place" := ("SqlData".data.rows[0].col[4]);
	                    "DB_RobotMission"."ZRot_Pick-Place" := ("SqlData".data.rows[0].col[5]);
	                    "DB_RobotMission".X_approach := ("SqlData".data.rows[0].col[6]);
	                    "DB_RobotMission".Y_approach := ("SqlData".data.rows[0].col[7]);
	                    "DB_RobotMission".Z_approach := ("SqlData".data.rows[0].col[8]);
	                    "DB_RobotMission".XRot_approach := ("SqlData".data.rows[0].col[9]);
	                    "DB_RobotMission".YRot_approach := ("SqlData".data.rows[0].col[10]);
	                    "DB_RobotMission".ZRot_approach := ("SqlData".data.rows[0].col[11]);
	                    //"DB_RobotMission".ApproachType := DINT_TO_INT("SqlData".data.rows[0].col[12]);
	                    "DB_RobotMission".ApproachType := "FC_ExtractApproach"(approachVal := "SqlData".data.rows[0].col[12], pick := FALSE);
	                    "DB_RobotMission".Object_Type := "Pallet";
	                    "DB_RobotMission".Unit_code := 10 + #MCRequested; //MC1-4 -> 11-14
	                    "DB_RobotMission".Gripper_code := #GripperRequested;
	                    "DB_RobotMission".Gripper_Side := 1;
	                    //"DB_RobotMission".Option
	                    "DB_executeQuery".readyForNextQuery := TRUE;

	                    #Dispatcher["_Pallet_MC_to_Robot"] := 40;
	                ELSIF "DB_executeQuery".dataError THEN
	                    //Errore
	                    "DB_executeQuery".readyForNextQuery := TRUE;
	                    #Error := 4099;
	                    #Dispatcher["_Pallet_MC_to_Robot"] := 4099;
	                END_IF;
	            40:
	                "DB_RobotMission".Command := "CMD_RobotPickObject";
	                IF "DB_RobotMissionStatus".StatusCode = "cmd_acquired" OR
	                    "DB_RobotMissionStatus".StatusCode = "cmd_executing" THEN
	                    #Dispatcher["_Pallet_MC_to_Robot"] := 50;
	                END_IF;
	            50:
	                IF "DB_RobotMissionStatus".StatusCode = "cmd_executed" THEN
	                    IF "DB_RobotMission".Gripper_Side = 2 THEN
	                        #GripperOccuped[2] := TRUE;
	                    ELSE
	                        #GripperOccuped[1] := TRUE;
	                    END_IF;
	                    "DB_RobotMission".Command := 0;  ///\\\

	                    // RAW, NON LOADED (18/9): il prelievo pallet dal magazzino
	                    // scrive RAW ("il pallet lo considero grezzo cosi' va in
	                    // macchina", 50 di Pallet_TRAY_to_Robot) e su quel valore sono
	                    // costruite le viste e i filtri del ciclo, che cercano STATUS=4.
	                    // Con LOADED=1 la riga a DB diceva uno stato che nessuno
	                    // interroga: il pallet in pinza risultava invisibile.
	                    #Dispatcher["updatePartOnRobot"] := 10 + DINT_TO_INT("RAW");

	                    #Dispatcher["_Pallet_MC_to_Robot"] := 60;
	                END_IF;
	            60:
	                IF #Dispatcher["updatePartOnRobot"] = 0 THEN
	                    #Dispatcher["updatePartOnMC"] := 30 + DINT_TO_INT("EMPTY");

	                    // IL PEZZO SI AZZERA SUBITO (18/9): senza il pallet in macchina
	                    // non c'e' niente che possa trattenere un pezzo — qualunque cosa
	                    // dica piecepresent, li' dentro e' vuoto. Visto in campo: pallet
	                    // smontato e registro ancora a 1033, il 50 di FB204 ha concluso
	                    // che c'era un finito da prelevare.
	                    IF #MCRequested = 1 THEN
	                        "DB_MC1".piecepresent[1] := 0;
	                    END_IF;

	                    // IL PALLET NO: il ramo 31..35 di updatePartOnMC lo legge per
	                    // sapere QUALE riga aggiornare a POS_PLANT=1000, e gira in una
	                    // REGION successiva dello stesso scan. Azzerarlo qui gli
	                    // toglierebbe il dato sotto i piedi. Si azzera al 70, a catena
	                    // chiusa.

	                    #Dispatcher["_Pallet_MC_to_Robot"] := 70;
	                END_IF;
	            70:
	                IF #Dispatcher["updatePartOnMC"] = 0 THEN
	                    // ADESSO il registro puo' cadere: la query lo ha gia' letto e
	                    // il database sa che il pallet e' a bordo.
	                    // IL REGISTRO DELLA MACCHINA VA AZZERATO (16/9): il pallet e'
	                    // appena uscito, ma DB_MC1.pallet restava al valore dichiarato.
	                    // Il 30 di FB204 confronta order.PALLET con quel registro per
	                    // decidere se montare il pallet: con il registro che mente,
	                    // saltava il montaggio e passava al check pinza chiedendo la
	                    // pinza del PEZZO.
	                    IF #MCRequested = 1 THEN
	                        "DB_MC1".pallet := 0;
	                    ELSIF #MCRequested = 2 THEN
	                        "DB_MC2".pallet := 0;
	                    END_IF;

	                    #Dispatcher["_Pallet_MC_to_Robot"] := 0;
	                END_IF;
	        END_CASE;
	    END_REGION

	END_REGION


	REGION PARTS_MANAGER
	    //abbasso velocita se ho i cassetti aperti? TODO
	    REGION Part_TRAY_to_Robot
	        CASE #Dispatcher["_Part_TRAY_to_Robot"] OF
	            0: //nothing to do
	                ;

	            10: //prepare mission data
	                IF "SqlCommands".sqlCommands[0] = '' THEN
	                    // Il magazzino deve essere abilitato: porta operatore chiusa e
	                    // registro cassetto coerente con i sensori. Senza questa guardia
	                    // la catena si fida di ExtractedTray, che e' Retain e puo' mentire.
	                    IF NOT "DB_BOX_1".Robot_enabled_to_work THEN
	                        #Error := 949;
	                        #Dispatcher["_Part_TRAY_to_Robot"] := 0;
	                    ELSIF #GripperOccuped[1] THEN
	                        //gripper not empty
	                        #Error := "_Part_TRAY_to_Robot" * 100 + 21;     //error 521
	                        #Dispatcher["_Part_TRAY_to_Robot"] := "_Part_TRAY_to_Robot" * 100 + 21;
	                    ELSIF NOT #RemoteMode AND #MCRequested = 0 THEN   // HMI: pezzo esplicito nel cassetto estratto
	                        #queryTemp := CONCAT(IN1 := 'select X_PICK,y_PICK,z_PICK,X_ROT,y_rot,Z_ROt,APPROACH_type,APPROACH_x,APPROACH_y,APPROACH_Z,cast(TRAY as int) from COORDINATES_PIECES_TRAYS_4Robot where TRAY = $'',
	                                             IN2 := "INT_TO_STRING_WITHOUT_SIGN"("DB_BOX_1".ExtractedTray),
	                                             IN3 := '$' AND SUB_POS=',
	                                             IN4 := "INT_TO_STRING_WITHOUT_SIGN"(#PartSubPos));
	                        #queryStartExecution := TRUE;

	                        #Dispatcher["_Part_TRAY_to_Robot"] := 20;
	                    ELSE
	                        // AUTOMATICO: SUB_POS in coda (col[11]) per congelare la tasca,
	                        // cosi' il finito potra' tornare esattamente da dove e' uscito.
	                        // FILTRO PER TIPO PEZZO (16/9): partType, non order_ID. Il
	                        // magazzino contiene grezzi di un tipo, non grezzi riservati
	                        // a un ordine — cosi' il rifornimento a meta' produzione viene
	                        // visto subito.
	                        // FILTRO SUL CASSETTO ESTRATTO (5/9): il CHECK CASSETTO di
	                        // FB204 (stati 40-46) garantisce che quando si arriva qui il
	                        // cassetto giusto e' gia' fuori.
	                        IF #MCRequested = 1 THEN
	                            #queryTemp := CONCAT(IN1 := 'select X_PICK,y_PICK,z_PICK,X_ROT,y_rot,Z_ROt,APPROACH_type,APPROACH_x,APPROACH_y,APPROACH_Z,cast(TRAY as int),SUB_POS from COORDINATES_PIECES_TRAYS_4Robot where STATUS=4 AND partType=',
	                                                 IN2 := "INT_TO_STRING_WITHOUT_SIGN"(DINT_TO_INT("DB_MC1".order.PIECE)),
	                                                 IN3 := ' AND TRAY=$'',
	                                                 IN4 := "INT_TO_STRING_WITHOUT_SIGN"("DB_BOX_1".ExtractedTray),
	                                                 IN5 := '$'');
	                        ELSE
	                            #queryTemp := CONCAT(IN1 := 'select X_PICK,y_PICK,z_PICK,X_ROT,y_rot,Z_ROt,APPROACH_type,APPROACH_x,APPROACH_y,APPROACH_Z,cast(TRAY as int),SUB_POS from COORDINATES_PIECES_TRAYS_4Robot where STATUS=4 AND partType=',
	                                                 IN2 := "INT_TO_STRING_WITHOUT_SIGN"(DINT_TO_INT("DB_MC2".order.PIECE)),
	                                                 IN3 := ' AND TRAY=$'',
	                                                 IN4 := "INT_TO_STRING_WITHOUT_SIGN"("DB_BOX_1".ExtractedTray),
	                                                 IN5 := '$'');
	                        END_IF;
	                        #queryStartExecution := TRUE;

	                        #Dispatcher["_Part_TRAY_to_Robot"] := 20;
	                    END_IF;
	                END_IF;

	            20:  //execute query
	                // PRESA IN CARICO VERIFICATA: non basta che il ponte sia occupato,
	                // deve esserci LA NOSTRA query. SqlData e' un buffer unico condiviso
	                // con FB204 e con le altre catene: senza questo confronto si puo'
	                // leggere la risposta di un altro richiedente (3/9: PartProgID
	                // 100000 al posto di 1, coordinate di approccio lette come dati).
	                IF NOT "DB_executeQuery".readyForNextQuery
	                    AND "SqlCommands".sqlCommands[0] = #queryTemp THEN
	                    #Dispatcher["_Part_TRAY_to_Robot"] := 30;
	                END_IF;

	            30:  // wait for result DB -> prepare mission data
	                IF "DB_executeQuery".dataReady AND "DB_executeQuery".noData THEN
	                    // Nessun pezzo trovato per quest'ordine. Con FB6 corretto
	                    // "zero righe" non e' piu' dataError, quindi va intercettato
	                    // qui: senza, si proseguirebbe con coordinate a zero.
	                    "DB_executeQuery".readyForNextQuery := true;
	                    #Error := 991;
	                    #Dispatcher["_Part_TRAY_to_Robot"] := 991;
	                ELSIF "DB_executeQuery".dataReady AND NOT "DB_executeQuery".dataError THEN

	                    IF ("SqlData".data.rows[0].col[10] = "DB_BOX_1".ExtractedTray) THEN
	                        //tray_requested is ready!
	                        "DB_RobotMission"."X_Pick-Place" := ("SqlData".data.rows[0].col[0]);
	                        "DB_RobotMission"."Y_Pick-Place" := ("SqlData".data.rows[0].col[1]);
	                        "DB_RobotMission"."Z_Pick-Place" := ("SqlData".data.rows[0].col[2]);
	                        "DB_RobotMission"."XRot_Pick-Place" := ("SqlData".data.rows[0].col[3]);
	                        "DB_RobotMission"."YRot_Pick-Place" := ("SqlData".data.rows[0].col[4]);
	                        "DB_RobotMission"."ZRot_Pick-Place" := ("SqlData".data.rows[0].col[5]);
	                        "DB_RobotMission".X_approach := ("SqlData".data.rows[0].col[7]);
	                        "DB_RobotMission".Y_approach := ("SqlData".data.rows[0].col[8]);
	                        "DB_RobotMission".Z_approach := ("SqlData".data.rows[0].col[9]);
	                        "DB_RobotMission".XRot_approach := 0;
	                        "DB_RobotMission".YRot_approach := 0;
	                        "DB_RobotMission".ZRot_approach := 0;
	                        "DB_RobotMission".ApproachType := "FC_ExtractApproach"(approachVal := "SqlData".data.rows[0].col[6], pick := TRUE);
	                        "DB_RobotMission".Object_Type := "Part";
	                        "DB_RobotMission".Unit_code := "Warehouse1";
	                        "DB_RobotMission".Gripper_Side := 1;
	                        "DB_RobotMission".Gripper_code := #GripperRequested;

	                        // congelo la tasca: il finito dovra' tornare qui
	                        IF #RemoteMode OR #MCRequested > 0 THEN
	                            #PartSubPos := DINT_TO_INT("SqlData".data.rows[0].col[11]);
	                        END_IF;

	                        "DB_executeQuery".readyForNextQuery := true;

	                        #Dispatcher["_Part_TRAY_to_Robot"] := 40;
	                    ELSE
	                        "DB_executeQuery".readyForNextQuery := true;
	                        #Tray_ID := DINT_TO_INT("SqlData".data.rows[0].col[10]);
	                        "DB_BOX_1".RequestedTray := DINT_TO_INT("SqlData".data.rows[0].col[10]);

	                        #Dispatcher["_Part_TRAY_to_Robot"] := 100;
	                    END_IF;
	                ELSIF "DB_executeQuery".dataError THEN
	                    "DB_executeQuery".readyForNextQuery := true;
	                    #Error := 991;
	                    #Dispatcher["_Part_TRAY_to_Robot"] := 991;
	                END_IF;

	            40:
	                "DB_RobotMission".Command := "CMD_RobotPickObject";
	                IF "DB_RobotMissionStatus".StatusCode = "cmd_acquired" OR
	                    "DB_RobotMissionStatus".StatusCode = "cmd_executing" THEN

	                    #Dispatcher["_Part_TRAY_to_Robot"] := 50;
	                END_IF;

	            50: // PRELIEVO CONCLUSO: CONFERMA COL SENSORE (16/9).
	                // Gripper1_Closed non dice "chele chiuse": il robot gestisce un
	                // extracorsa e se non ha afferrato niente le riapre. Chiuse =
	                // PEZZO A BORDO. Finora la catena si fidava del solo cmd_executed
	                // e scriveva "grezzo prelevato" su un prelievo che poteva non
	                // essere avvenuto — poi tutto il ciclo proseguiva su quel dato.
	                IF "DB_RobotMissionStatus".StatusCode = "cmd_executed" THEN
	                    IF "Gripper1_Closed" THEN
	                        // preso davvero
	                        #retryPick := FALSE;
	                        #GripperOccuped[1] := TRUE;
	                        "DB_RobotMission".Command := 0;  ///\\\
	                        #Dispatcher["updatePartOnRobot"] := 10 + DINT_TO_INT("RAW");

	                        #Dispatcher["_Part_TRAY_to_Robot"] := 60;

	                    ELSIF NOT #retryPick THEN
	                        // PRIMO FALLIMENTO: la tasca era vuota. Lo dico al database
	                        // — e' la verita', li' non c'era niente — e rilancio dal 10.
	                        // La query rifara' la ricerca e trovera' la PROSSIMA tasca
	                        // grezza dello stesso cassetto, senza bisogno di una query
	                        // diversa: marcare la tasca corregge il magazzino E fa
	                        // avanzare la scelta, con un gesto solo.
	                        #retryPick := TRUE;
	                        "DB_RobotMission".Command := 0;  ///\\\
	                        #Dispatcher["_Part_TRAY_to_Robot"] := 55;

	                    ELSE
	                        // SECONDO FALLIMENTO CONSECUTIVO: non e' una tasca vuota,
	                        // e' un problema. Cella in HOLD e allarme, senza muovere il
	                        // robot: la messa in sicurezza la fa l'operatore, che prima
	                        // guarda cosa e' successo.
	                        "DB_RobotMission".Command := 0;  ///\\\
	                        #retryPick := FALSE;
	                        #HOLD := TRUE;
	                        #Error := 992;                    // prelievo cassetto fallito due volte
	                        "DB_MC1".Dispatcher["_master"] := 9999;
	                        #MissionCode := 0;
	                        #Dispatcher["_Part_TRAY_to_Robot"] := 0;
	                    END_IF;
	                END_IF;

	            55: // marca vuota la tasca fallita, poi rilancia il prelievo
	                IF "SqlCommands".sqlCommands[0] = '' THEN
	                    #queryTemp := CONCAT(IN1 := 'UPDATE [POSITION] SET STATUS=2 WHERE PARENT=$'TRAY_',
	                                         IN2 := "INT_TO_STRING_WITHOUT_SIGN"("DB_BOX_1".ExtractedTray),
	                                         IN3 := '$' AND SUB_POS=',
	                                         IN4 := "INT_TO_STRING_WITHOUT_SIGN"(#PartSubPos));
	                    #queryStartExecution := TRUE;
	                    #Dispatcher["_Part_TRAY_to_Robot"] := 56;
	                END_IF;

	            56: // presa in carico VERIFICATA
	                IF NOT "DB_executeQuery".readyForNextQuery
	                    AND "SqlCommands".sqlCommands[0] = #queryTemp THEN
	                    #Dispatcher["_Part_TRAY_to_Robot"] := 57;
	                END_IF;

	            57: // tasca marcata: riparto dal 10, la query trovera' la prossima
	                IF "DB_executeQuery".dataReady THEN
	                    "DB_executeQuery".readyForNextQuery := TRUE;
	                    #queryTemp := '';
	                    #queryStartExecution := FALSE;
	                    "FC_MQTT"(insert := true,
	                              send := false,
	                              topic := 'FROM_PLANT/DECLARE/TRAY',
	                              payload := STRING_TO_WSTRING(CONCAT(IN1 := "INT_TO_STRING_WITHOUT_SIGN"("DB_BOX_1".ExtractedTray),
	                                                                                               IN2 := ';',
	                                                                                               IN3 := "INT_TO_STRING_WITHOUT_SIGN"(#PartSubPos),
	                                                                                               IN4 := ';2')));
	                    #Dispatcher["_Part_TRAY_to_Robot"] := 10;
	                END_IF;

	            60:  // updateDB
	                IF #Dispatcher["updatePartOnRobot"] = 0 THEN
	                    #Dispatcher["updatePartOnTray"] := 10 + DINT_TO_INT("EMPTY");

	                    #Dispatcher["_Part_TRAY_to_Robot"] := 70;
	                END_IF;
	            70:
	                IF #Dispatcher["updatePartOnTray"] = 0 THEN
	                    #retryPick := FALSE;
	                    #Dispatcher["_Part_TRAY_to_Robot"] := 0;
	                END_IF;

	            100: //////////////// SPECIAL CONDITION ////////////////
	                //wait the right tray is ready -> restart this mission
	                IF "DB_BOX_1".ExtractedTray = #Tray_ID THEN
	                    #MissionCode := 0;      //da controllare...

	                    #Dispatcher["_Part_TRAY_to_Robot"] := 10;
	                END_IF;

	        END_CASE;
	    END_REGION

	    REGION Part_Robot_to_TRAY
	        CASE #Dispatcher["_Part_Robot_to_TRAY"] OF
	            0: //nothing to do
	                ;
	            10: //prepare mission data
	                IF "SqlCommands".sqlCommands[0] = '' THEN
	                    IF NOT "DB_BOX_1".Robot_enabled_to_work THEN
	                        #Error := 949;
	                        #Dispatcher["_Part_Robot_to_TRAY"] := 0;
	                    ELSIF NOT #GripperOccuped[1] AND NOT #GripperOccuped[2] THEN
	                        //gripper EMPTY
	                        #Error := "_Part_Robot_to_TRAY" * 100 + 21;     //error 621
	                        #Dispatcher["_Part_Robot_to_TRAY"] := "_Part_Robot_to_TRAY" * 100 + 21;
	                    ELSE
	                        IF NOT #RemoteMode AND #PartSubPos > 0 THEN   // HMI: posizione esplicita
	                            #queryTemp := CONCAT(IN1 := 'select X_PICK,y_PICK,z_PICK,X_ROT,y_rot,Z_ROt,APPROACH_type,APPROACH_x,APPROACH_y,APPROACH_Z from COORDINATES_PIECES_TRAYS_4Robot where TRAY = $'',
	                                                 IN2 := "INT_TO_STRING_WITHOUT_SIGN"(#Tray_ID),
	                                                 IN3 := '$' AND SUB_POS=',
	                                                 IN4 := "INT_TO_STRING_WITHOUT_SIGN"(#PartSubPos));
	                        ELSIF NOT #RemoteMode THEN   // HMI: prima vuota — SUB_POS in coda (col[10]) per l'update stati
	                            #queryTemp := CONCAT(IN1 := 'select X_PICK,y_PICK,z_PICK,X_ROT,y_rot,Z_ROt,APPROACH_type,APPROACH_x,APPROACH_y,APPROACH_Z,SUB_POS from COORDINATES_PIECES_TRAYS_4Robot where TRAY = $'',
	                                                 IN2 := "INT_TO_STRING_WITHOUT_SIGN"(#Tray_ID),
	                                                 IN3 := '$' AND STATUS=2');  //empty
	                        ELSE
	                            // AUTOMATICO: il lato 2 porta il FINITO uscito dalla macchina,
	                            // che torna nella tasca del suo grezzo (PartSubPosMC).
	                            // Il lato 1 porta un grezzo mai entrato: tasca corrente.
	                            IF #GripperOccuped[2] AND #Gripper_ID[2] > 0 THEN
	                                #temp := #PartSubPosMC;
	                            ELSE
	                                #temp := #PartSubPos;
	                            END_IF;
	                            #queryTemp := CONCAT(IN1 := 'select X_PICK,y_PICK,z_PICK,X_ROT,y_rot,Z_ROt,APPROACH_type,APPROACH_x,APPROACH_y,APPROACH_Z from COORDINATES_PIECES_TRAYS_4Robot where TRAY = $'',
	                                                 IN2 := "INT_TO_STRING_WITHOUT_SIGN"(#Tray_ID),
	                                                 IN3 := '$' AND SUB_POS=',
	                                                 IN4 := "INT_TO_STRING_WITHOUT_SIGN"(#temp));
	                        END_IF;
	                        #queryStartExecution := TRUE;

	                        #Dispatcher["_Part_Robot_to_TRAY"] := 20;
	                    END_IF;
	                END_IF;

	            20:  //execute query
	                // PRESA IN CARICO VERIFICATA: SqlData e' un buffer unico condiviso,
	                // senza il confronto su sqlCommands[0] si legge la risposta di un
	                // altro richiedente.
	                IF NOT "DB_executeQuery".readyForNextQuery
	                    AND "SqlCommands".sqlCommands[0] = #queryTemp THEN
	                    #Dispatcher["_Part_Robot_to_TRAY"] := 30;
	                END_IF;

	            30:  // wait for result DB -> prepare mission data
	                IF "DB_executeQuery".dataReady AND "DB_executeQuery".noData THEN
	                    // tasca di destinazione non trovata: con FB6 corretto "zero righe"
	                    // non e' piu' dataError, va intercettato qui.
	                    "DB_executeQuery".readyForNextQuery := true;
	                    #Error := "_Part_Robot_to_TRAY" * 100 + 91;         //Error 691
	                    #Dispatcher["_Part_Robot_to_TRAY"] := "_Part_Robot_to_TRAY" * 100 + 91;
	                ELSIF "DB_executeQuery".dataReady AND NOT "DB_executeQuery".dataError THEN
	                    "DB_RobotMission"."X_Pick-Place" := ("SqlData".data.rows[0].col[0]);
	                    "DB_RobotMission"."Y_Pick-Place" := ("SqlData".data.rows[0].col[1]);
	                    "DB_RobotMission"."Z_Pick-Place" := ("SqlData".data.rows[0].col[2]);
	                    "DB_RobotMission"."XRot_Pick-Place" := ("SqlData".data.rows[0].col[3]);
	                    "DB_RobotMission"."YRot_Pick-Place" := ("SqlData".data.rows[0].col[4]);
	                    "DB_RobotMission"."ZRot_Pick-Place" := ("SqlData".data.rows[0].col[5]);
	                    "DB_RobotMission".X_approach := ("SqlData".data.rows[0].col[7]);
	                    "DB_RobotMission".Y_approach := ("SqlData".data.rows[0].col[8]);
	                    "DB_RobotMission".Z_approach := ("SqlData".data.rows[0].col[9]);
	                    "DB_RobotMission".XRot_approach := 0;
	                    "DB_RobotMission".YRot_approach := 0;
	                    "DB_RobotMission".ZRot_approach := 0;
	                    //"DB_RobotMission".ApproachType := DINT_TO_INT("SqlData".data.rows[0].col[6]);
	                    "DB_RobotMission".ApproachType := "FC_ExtractApproach"(approachVal := "SqlData".data.rows[0].col[6], pick := FALSE);
	                    "DB_RobotMission".Object_Type := "Part";
	                    "DB_RobotMission".Unit_code := "Warehouse1";
	                    IF #Gripper_ID[2] > 0 AND #GripperOccuped[2] THEN
	                        "DB_RobotMission".Gripper_Side := 2;
	                    ELSE
	                        "DB_RobotMission".Gripper_Side := 1;
	                    END_IF;

	                    //"DB_RobotMission".Option
	                    //#BoxRequested :=
	                    IF NOT #RemoteMode AND #PartSubPos <= 0 THEN
	                        // posizione scelta dalla query "prima vuota": congelata per l'update stati
	                        #PartSubPos := DINT_TO_INT("SqlData".data.rows[0].col[10]);
	                    END_IF;

	                    "DB_executeQuery".readyForNextQuery := true;

	                    #Dispatcher["_Part_Robot_to_TRAY"] := 40;
	                ELSIF "DB_executeQuery".dataError THEN
	                    "DB_executeQuery".readyForNextQuery := true;

	                    #Error := "_Part_Robot_to_TRAY" * 100 + 91;         //Error 691
	                    #Dispatcher["_Part_Robot_to_TRAY"] := "_Part_Robot_to_TRAY" * 100 + 91;
	                END_IF;
	            40:
	                "DB_RobotMission".Command := "CMD_RobotPlaceObject";
	                IF "DB_RobotMissionStatus".StatusCode = "cmd_acquired" OR
	                    "DB_RobotMissionStatus".StatusCode = "cmd_executing" THEN

	                    #Dispatcher["_Part_Robot_to_TRAY"] := 50;
	                END_IF;
	            50:
	                IF "DB_RobotMissionStatus".StatusCode = "cmd_executed" THEN
	                    "DB_RobotMission".Command := 0;  ///\\\

	                    #Dispatcher["updatePartOnRobot"] := 10 + DINT_TO_INT("EMPTY");
	                    #GripperOccuped["DB_RobotMission".Gripper_Side] := FALSE;

	                    #Dispatcher["_Part_Robot_to_TRAY"] := 60;
	                END_IF;
	            60:  // updateDB
	                IF #Dispatcher["updatePartOnRobot"] = 0 THEN
	                    #Dispatcher["updatePartOnTray"] := 10 + DINT_TO_INT("FINISHED");

	                    #Dispatcher["_Part_Robot_to_TRAY"] := 70;
	                END_IF;
	            70:
	                IF #Dispatcher["updatePartOnTray"] = 0 THEN
	                    #Dispatcher["_Part_Robot_to_TRAY"] := 0;
	                END_IF;


	        END_CASE;
	    END_REGION

	    REGION Part_Robot_to_MC
	        CASE #Dispatcher["_Part_Robot_to_MC"] OF
	            0: //nothing to do
	                ;

	            10: //prepare mission data
	                IF "SqlCommands".sqlCommands[0] = '' THEN
	                    IF NOT #GripperOccuped[1] AND NOT #GripperOccuped[2] THEN
	                        //gripper empty
	                        #Error := 22;
	                        #Dispatcher["_Part_Robot_to_MC"] := 7001;
	                    ELSE
	                        // QUOTE DALLA VISTA COORDINATES_Z_MC (19/9): il calcolo
	                        // Z era scritto a mano qui, nel 10 di Part_MC_to_Robot e
	                        // dentro COORDINATES_PICKPLACE_MC — tre copie della
	                        // stessa formula, tre occasioni di divergenza.
	                        // E la geometria delle ganasce era INGLOBATA in FIXTURE.Z:
	                        // cambiando le chele il pezzo finiva alla quota delle
	                        // vecchie, 2,3 mm troppo in basso sulla morsa.
	                        // Adesso FIXTURE.Z e' pallet piu' corpo morsa senza chele,
	                        // e la vista aggiunge Z_CLAW - Z_SINK_CLAW.
	                        // Z_PLACE_MC = deposito del GREZZO (qui si deposita).
	                        #queryTemp := 'select P.X,P.Y,Z.Z_PLACE_MC,P.X_ROT,P.Y_ROT,P.Z_ROT,P.APPROACH_TYPE,P.APPROACH_X,P.APPROACH_Y,P.APPROACH_Z from POSITION P,COORDINATES_Z_MC Z where P.PARENT=$'MC_1$' and ';
	                        IF #RemoteMode THEN
	                            IF #MCRequested = 1 AND "DB_MC1".order.ID > 0 THEN
	                                #queryTemp := CONCAT(IN1 := #queryTemp,
	                                                     IN2 := 'Z.ORDER_ID=',
	                                                     IN3 := "INT_TO_STRING_WITHOUT_SIGN"(DINT_TO_INT("DB_MC1".order.ID)));
	                            ELSE
	                                #Error := 936;   // deposito auto senza ordine attivo
	                            END_IF;
	                        ELSE
	                            // MANUALE (30): ordine attivo se presente, altrimenti il piu' recente
	                            IF "DB_MC1".order.ID > 0 THEN
	                                #queryTemp := CONCAT(IN1 := #queryTemp,
	                                                     IN2 := 'Z.ORDER_ID=',
	                                                     IN3 := "INT_TO_STRING_WITHOUT_SIGN"(DINT_TO_INT("DB_MC1".order.ID)));
	                            ELSE
	                                #queryTemp := CONCAT(IN1 := #queryTemp,
	                                                     IN2 := 'Z.MC=1 order by Z.ORDER_ID desc');
	                            END_IF;
	                        END_IF;

	                        IF #Error = 0 THEN
	                            #queryStartExecution := TRUE;
	                            #Dispatcher["_Part_Robot_to_MC"] := 20;
	                        END_IF;
	                    END_IF;
	                END_IF;

	            20:  //execute query
	                // PRESA IN CARICO VERIFICATA: SqlData e' un buffer unico condiviso,
	                // senza il confronto su sqlCommands[0] si legge la risposta di un
	                // altro richiedente — qui sarebbero le QUOTE DI DEPOSITO in macchina.
	                IF NOT "DB_executeQuery".readyForNextQuery
	                    AND "SqlCommands".sqlCommands[0] = #queryTemp THEN
	                    #Dispatcher["_Part_Robot_to_MC"] := 30;
	                END_IF;

	            30:  // wait for result DB -> prepare mission data
	                IF "DB_executeQuery".dataReady AND "DB_executeQuery".noData THEN
	                    // quote di deposito non trovate (ordine/pezzo/attrezzatura non
	                    // coerenti a DB): con FB6 corretto va intercettato qui.
	                    "DB_executeQuery".readyForNextQuery := true;
	                    #Error := "_Part_Robot_to_MC" * 100 + 99;           //error 799
	                    #Dispatcher["_Part_Robot_to_MC"] := "_Part_Robot_to_MC" * 100 + 99;
	                ELSIF "DB_executeQuery".dataReady AND NOT "DB_executeQuery".dataError THEN

	                    "DB_RobotMission"."X_Pick-Place" := ("SqlData".data.rows[0].col[0]);
	                    "DB_RobotMission"."Y_Pick-Place" := ("SqlData".data.rows[0].col[1]);
	                    "DB_RobotMission"."Z_Pick-Place" := ("SqlData".data.rows[0].col[2]);
	                    "DB_RobotMission"."XRot_Pick-Place" := ("SqlData".data.rows[0].col[3]);
	                    "DB_RobotMission"."YRot_Pick-Place" := ("SqlData".data.rows[0].col[4]);
	                    "DB_RobotMission"."ZRot_Pick-Place" := ("SqlData".data.rows[0].col[5]);
	                    "DB_RobotMission".X_approach := ("SqlData".data.rows[0].col[7]);
	                    "DB_RobotMission".Y_approach := ("SqlData".data.rows[0].col[8]);
	                    "DB_RobotMission".Z_approach := ("SqlData".data.rows[0].col[9]);
	                    "DB_RobotMission".XRot_approach := 0;
	                    "DB_RobotMission".YRot_approach := 0;
	                    "DB_RobotMission".ZRot_approach := 0;
	                    //"DB_RobotMission".ApproachType := DINT_TO_INT("SqlData".data.rows[0].col[6]);
	                    "DB_RobotMission".ApproachType := "FC_ExtractApproach"(approachVal := "SqlData".data.rows[0].col[6], pick := FALSE);
	                    "DB_RobotMission".Object_Type := "Part";
	                    "DB_RobotMission".Unit_code := #MCRequested + 10;
	                    "DB_RobotMission".Gripper_code := #GripperRequested;
	                    "DB_RobotMission".Gripper_Side := 1;
	                    //"DB_RobotMission".Option

	                    "DB_executeQuery".readyForNextQuery := true;

	                    // SPINTA IN BATTUTA: seconda lettura, sulla vista COORDINATES_PUSH_MC.
	                    // Si legge QUI, PRIMA di lanciare la missione, e si congela: il
	                    // robot non deve mai aspettare il ponte SQL con le chele chiuse
	                    // accanto a un pezzo posato. Da questo punto in poi un cambio a
	                    // database non ha effetto fino al pezzo successivo.
	                    #xPushTemp := 0;
	                    #xStopTemp := 0;
	                    #Dispatcher["_Part_Robot_to_MC"] := 32;
	                ELSIF "DB_executeQuery".dataError THEN
	                    //Errore
	                    #Error := "_Part_Robot_to_MC" * 100 + 99;           //error 799
	                    #Dispatcher["_Part_Robot_to_MC"] := "_Part_Robot_to_MC" * 100 + 99;
	                    "DB_executeQuery".readyForNextQuery := true;
	                END_IF;

	            32:  // SPINTA: compone la query sulle quote di spinta e arrivo.
	                // Vale anche in MANUALE (comando 30 dal pannello): si usa l'ordine
	                // attivo se c'e', altrimenti il piu' recente, come fa il 10 per le
	                // quote di deposito.
	                IF #MCRequested <> 1 THEN
	                    // MC2 non esiste in questa cella: nessuna spinta
	                    #Dispatcher["_Part_Robot_to_MC"] := 40;
	                ELSIF "SqlCommands".sqlCommands[0] = '' THEN
	                    IF "DB_MC1".order.ID > 0 THEN
	                        #queryTemp := CONCAT(IN1 := 'select X_PUSH,X_STOP from COORDINATES_PUSH_MC where MC=1 and ORDER_ID=',
	                                             IN2 := "INT_TO_STRING_WITHOUT_SIGN"(DINT_TO_INT("DB_MC1".order.ID)));
	                    ELSE
	                        // nessun ordine attivo: il piu' recente, come il 10
	                        #queryTemp := 'select top 1 X_PUSH,X_STOP from COORDINATES_PUSH_MC where MC=1 order by ORDER_ID desc';
	                    END_IF;
	                    #queryStartExecution := TRUE;
	                    #Dispatcher["_Part_Robot_to_MC"] := 34;
	                END_IF;

	            34:  // presa in carico VERIFICATA della query spinta
	                IF NOT "DB_executeQuery".readyForNextQuery
	                    AND "SqlCommands".sqlCommands[0] = #queryTemp THEN
	                    #Dispatcher["_Part_Robot_to_MC"] := 36;
	                END_IF;

	            36:  // esito spinta. Le quote sono NULL quando la vista dice che la
	                // spinta non e' configurata, disabilitata, o il pezzo non ci sta.
	                // ATTENZIONE: il ponte SQL NON converte NULL in zero — restituisce
	                // valori casuali (visto 15/9: xStopTemp a -1.056.960.259 con
	                // PUSH_STATUS DISABLED). Quindi non ci si puo' fidare del valore:
	                // va verificato che sia PLAUSIBILE rispetto alla quota di deposito.
	                // Spinta e arrivo stanno per costruzione entro qualche centinaio di
	                // millimetri da X_PLACE: fuori da mezzo metro il dato e' spazzatura
	                // e la spinta non si fa.
	                IF "DB_executeQuery".dataReady THEN
	                    IF "DB_executeQuery".noData OR "DB_executeQuery".dataError THEN
	                        #xPushTemp := 0;
	                        #xStopTemp := 0;
	                    ELSE
	                        #xPushTemp := "SqlData".data.rows[0].col[0];
	                        #xStopTemp := "SqlData".data.rows[0].col[1];

	                        // controllo di plausibilita': entrambe le quote devono
	                        // stare entro 500 mm dalla quota di deposito appena letta
	                        IF ABS(#xPushTemp - "DB_RobotMission"."X_Pick-Place") > 500000
	                            OR ABS(#xStopTemp - "DB_RobotMission"."X_Pick-Place") > 500000
	                        THEN
	                            #xPushTemp := 0;
	                            #xStopTemp := 0;
	                        END_IF;
	                    END_IF;
	                    "DB_executeQuery".readyForNextQuery := TRUE;
	                    #queryTemp := '';
	                    #queryStartExecution := FALSE;
	                    #Dispatcher["_Part_Robot_to_MC"] := 37;
	                END_IF;

	            37:  // SOFFIAGGIO: lunghezza chele morsa, larghezza pezzo e quota di
	                // appoggio verso il robot (19/9). Il robotista le legge prima di
	                // soffiare, in deposito e in prelievo.
	                // Query SEPARATA dalle quote: quelle sono critiche e passano da
	                // viste collaudate, queste servono a un soffiaggio e non devono
	                // appesantirle.
	                // VISTA DEDICATA (COORDINATES_BLOW_MC): la query coi join scritti
	                // a mano faceva 298 caratteri e queryTemp ne regge 254 — sarebbe
	                // arrivata troncata, come il 13599 del 15/9. Con la vista sono 96.
	                // Le tre variabili PROFINET NON si azzerano mai: restano quelle
	                // dell'ultimo pezzo finche' un nuovo giro non le sovrascrive. Se
	                // la query fallisce si prosegue coi valori vecchi — fermare la
	                // cella per una misura di soffiaggio sarebbe sproporzionato.
	                IF "SqlCommands".sqlCommands[0] = '' THEN
	                    IF "DB_MC1".order.ID > 0 THEN
	                        #queryTemp := CONCAT(IN1 := 'select CLAW_LENGTH,PART_WIDTH,STOP_BEYOND_CLAW from COORDINATES_BLOW_MC where ORDER_ID=',
	                                             IN2 := "INT_TO_STRING_WITHOUT_SIGN"(DINT_TO_INT("DB_MC1".order.ID)));
	                        #queryStartExecution := TRUE;
	                        #Dispatcher["_Part_Robot_to_MC"] := 38;
	                    ELSE
	                        // nessun ordine attivo (comando manuale): niente da leggere,
	                        // il robot usa i valori del giro precedente
	                        #Dispatcher["_Part_Robot_to_MC"] := 40;
	                    END_IF;
	                END_IF;

	            38:  // presa in carico VERIFICATA
	                IF NOT "DB_executeQuery".readyForNextQuery
	                    AND "SqlCommands".sqlCommands[0] = #queryTemp THEN
	                    #Dispatcher["_Part_Robot_to_MC"] := 39;
	                END_IF;

	            39:  // esito: scrive le tre variabili PROFINET.
	                // APPOGGIO COME MISURA, NON COME QUOTA (19/9): il robotista non
	                // vuole piu' la posizione X del pezzo, che calcola per conto suo —
	                // gli serve solo di quanto il pezzo appoggia, cioe' meta' ganascia
	                // piu' il tratto oltre la ganascia dichiarato a pannello.
	                // L'espressione e' tutta DInt (le colonne SqlData lo sono), quindi
	                // la somma in micron non trabocca e la conversione a Int avviene
	                // una volta sola sul risultato in mm.
	                // I micron del database diventano mm interi: per un soffiaggio il
	                // decimo non serve, e il robotista ha chiesto Int.
	                IF "DB_executeQuery".dataReady THEN
	                    IF NOT "DB_executeQuery".noData AND NOT "DB_executeQuery".dataError THEN
	                        "Vice_ClawLength_mm" := DINT_TO_INT("SqlData".data.rows[0].col[0] / 1000);
	                        "Part_Width_mm" := DINT_TO_INT("SqlData".data.rows[0].col[1] / 1000);
	                        "X_Support_mm" := DINT_TO_INT(("SqlData".data.rows[0].col[0] / 2
	                                                                                    + "SqlData".data.rows[0].col[2]) / 1000);
	                    END_IF;
	                    "DB_executeQuery".readyForNextQuery := TRUE;
	                    #queryTemp := '';
	                    #queryStartExecution := FALSE;
	                    #Dispatcher["_Part_Robot_to_MC"] := 40;
	                END_IF;

	            40:
	                // Il consenso alla spinta va alzato PRIMA del comando: il robot lo
	                // legge quando acquisisce la missione e sa se dovra' chiedere le
	                // due fasi in piu'. Quote a zero = deposito normale, come oggi.
	                "Q_PushEnable_MC" := (#xPushTemp <> 0) AND (#xStopTemp <> 0);
	                "Ok_PushSpinta_MC" := FALSE;
	                "Ok_PushArrivo_MC" := FALSE;

	                "DB_RobotMission".Command := "CMD_RobotPlaceObject";
	                IF "DB_RobotMissionStatus".StatusCode = "cmd_acquired" OR
	                    "DB_RobotMissionStatus".StatusCode = "cmd_executing" THEN
	                    IF "Q_PushEnable_MC" THEN
	                        #Dispatcher["_Part_Robot_to_MC"] := 42;
	                    ELSE
	                        #Dispatcher["_Part_Robot_to_MC"] := 50;
	                    END_IF;
	                END_IF;

	            42:  // SPINTA fase 1: il robot ha depositato e chiede la quota di spinta.
	                // HANDSHAKE BIDIREZIONALE concordato col robotista: il robot alza
	                // il bit, il PLC risponde col consenso, il robot ABBASSA il bit,
	                // il PLC abbassa il consenso. Solo allora la fase e' chiusa.
	                IF "Robot_PushDepositoFatto_MC" THEN
	                    "DB_RobotMission"."X_Pick-Place" := #xPushTemp;
	                    "Ok_PushSpinta_MC" := TRUE;
	                    #Dispatcher["_Part_Robot_to_MC"] := 43;
	                END_IF;

	            43:  // attesa che il robot abbassi il suo bit: ha letto la quota
	                IF NOT "Robot_PushDepositoFatto_MC" THEN
	                    "Ok_PushSpinta_MC" := FALSE;
	                    #Dispatcher["_Part_Robot_to_MC"] := 44;
	                END_IF;

	            44:  // SPINTA fase 2: il robot e' in posizione e chiede la quota di arrivo
	                IF "Robot_PushInPos_MC" THEN
	                    "DB_RobotMission"."X_Pick-Place" := #xStopTemp;
	                    "Ok_PushArrivo_MC" := TRUE;
	                    #Dispatcher["_Part_Robot_to_MC"] := 45;
	                END_IF;

	            45:  // attesa che il robot abbassi il suo bit: ha letto la quota
	                IF NOT "Robot_PushInPos_MC" THEN
	                    "Ok_PushArrivo_MC" := FALSE;
	                    #Dispatcher["_Part_Robot_to_MC"] := 50;
	                END_IF;

	            50:
	                IF "DB_RobotMissionStatus".StatusCode = "cmd_executed" OR
	                    "DB_RobotMissionStatus".StatusCode = "cmd_waitingNewCmd" THEN
	                    "DB_RobotMission".Command := 0;  ///\\\
	                    #GripperOccuped[1] := FALSE;

	                    // CORSA DELLA SPINTA applicata a QUESTO pezzo: il prelievo
	                    // dovra' andare a prenderlo dove la spinta lo ha portato, non
	                    // dove il deposito lo aveva messo. Zero se la spinta non c'e'
	                    // stata. Si azzera solo quando il pezzo esce dalla macchina.
	                    IF "Q_PushEnable_MC" THEN
	                        #xPushOffsetMC := #xStopTemp - #xPushTemp;
	                    ELSE
	                        #xPushOffsetMC := 0;
	                    END_IF;

	                    // consensi spinta abbassati a fine missione
	                    "Q_PushEnable_MC" := FALSE;
	                    "Ok_PushSpinta_MC" := FALSE;
	                    "Ok_PushArrivo_MC" := FALSE;

	                    // LA TASCA, IL CASSETTO E L'ORDINE del grezzo appena caricato
	                    // seguono il pezzo in macchina: il finito che ne uscira' dovra'
	                    // tornare esattamente li', e appartiene all'ordine che lo ha
	                    // lavorato.
	                    // IL CASSETTO E' NUOVO (16/9): prima TrayIdMC si scriveva solo
	                    // al deposito del finito, quindi per tutto il tempo in cui il
	                    // pezzo era in macchina puntava al cassetto PRECEDENTE. Al
	                    // cambio cassetto la UPDATE del finito finiva sul cassetto
	                    // vecchio e il pezzo non veniva registrato (visto 16/9: 16
	                    // prodotti, 15 tasche marcate finite). In piu' il 50 di FB204
	                    // rifiutava la missione 16, perche' la sua guardia chiede
	                    // TrayIdMC = ExtractedTray: al cambio cassetto ripiegava sulla
	                    // sequenza in due tempi (13 + 12) invece dell'ingresso unico.
	                    //
	                    // L'ORDINE E' NUOVO (18/9): col ciclo a missione 16 il finito
	                    // viene depositato nel giro SUCCESSIVO, e sull'ultimo pezzo di
	                    // un ordine il 102 di FB204 puo' aver gia' riallineato order.ID
	                    // a quello dopo. Senza congelarlo, quel pezzo verrebbe contato
	                    // all'ordine sbagliato: uno in meno al vecchio, uno in piu' al
	                    // nuovo, sempre sull'ultimo pezzo.
	                    #PartSubPosMC := #PartSubPos;
	                    #TrayIdMC := #Tray_ID;
	                    IF #MCRequested = 2 THEN
	                        #OrderIdMC := DINT_TO_INT("DB_MC2".order.ID);
	                    ELSE
	                        #OrderIdMC := DINT_TO_INT("DB_MC1".order.ID);
	                    END_IF;

	                    #Dispatcher["updatePartOnRobot"] := 10 + DINT_TO_INT("RAW");

	                    #Dispatcher["_Part_Robot_to_MC"] := 60;
	                END_IF;

	            60:
	                IF #Dispatcher["updatePartOnRobot"] = 0 THEN
	                    #Dispatcher["updatePartOnMC"] := 10 + DINT_TO_INT("RAW");

	                    #Dispatcher["_Part_Robot_to_MC"] := 70;
	                END_IF;

	            70:
	                IF #Dispatcher["updatePartOnMC"] = 0 THEN

	                    #Dispatcher["_Part_Robot_to_MC"] := 0;
	                END_IF;
	        END_CASE;
	    END_REGION

